Omron CX-Programmer project NewProject (CX-Programmer 9.74)

# PLC GERAL: CJ2M CPU33
I/O table (CPU CJ2M-CPU33): rack 0 slot 0 CJ1W-SCU21; rack 0 slot 1 CJ1W-DRM21; rack 0 slot 2 CJ1W-ID211; rack 0 slot 3 CJ1W-OC211; rack 0 slot 4 CJ1W-MAD42; rack 0 slot 11 CJ2M-EIP21

## Data types
TYPE s_equip_ios : STRUCT  (* Equipamento - Entradas *)
  om : BOOL;  (* Ordem de marcha *)
  oma : BOOL;  (* Ordem de abrir *)
  omf : BOOL;  (* Ordem de fechar *)
  rm : BOOL;  (* Resposta de marcha *)
  fca : BOOL;  (* Fim de curso aberta *)
  fcf : BOOL;  (* Fim de curso fechada *)
  de : BOOL;  (* Defeito electrico *)
  pf_bmb : BOOL;  (* Pulsos de funcionamento da bomba *)
END_STRUCT END_TYPE
TYPE s_equip_bits : STRUCT  (* Equipamento - Bits auxiliares *)
  s_aut : BOOL;  (* Automatico *)
  mdp : BOOL;  (* Disponibilidade *)
  ndp : BOOL;  (* Não disponivel *)
  dgm : BOOL;  (* Defeito geral de maquina *)
  rst : BOOL;  (* Reset *)
  cfa : BOOL;  (* Condição de funcionamento automatico *)
  cfm : BOOL;  (* Condição de funcionamento manual *)
  cfaa : BOOL;  (* Condição de funcionamento automatico abrir *)
  cfaf : BOOL;  (* Condição de funcionamento automatico fechar *)
  cfma : BOOL;  (* Condição de funcionamento manual abrir *)
  cfmf : BOOL;  (* Condição de funcionamento manual fechar *)
  st_hmi : BOOL;  (* Arranque HMI *)
  sp_hmi : BOOL;  (* Paragem HMI *)
  p_hmi : BOOL;  (* Pausa HMI *)
END_STRUCT END_TYPE
TYPE s_equip_defs : STRUCT  (* Equipamentos - Defeitos *)
  fm : BOOL;  (* Falha de marcha *)
  fma : BOOL;  (* Falha de manobra abrir *)
  fmf : BOOL;  (* Falha de manobra fechar *)
  de : BOOL;  (* Defeito electrico *)
  dv : BOOL;  (* Deposito vazio *)
END_STRUCT END_TYPE
TYPE s_equip : STRUCT  (* Equipamento *)
  ios : s_equip_ios;  (* Entradas *)
  bits : s_equip_bits;  (* Bits *)
  defs : s_equip_defs;  (* Defeitos *)
  es : INT;  (* Estado *)
  tm_b : INT;  (* Tempo entre bombagens *)
  rsv1 : INT Dimensions=[5];  (* Reserva *)
END_STRUCT END_TYPE
TYPE s_deposito_p : STRUCT  (* Deposito de produto *)
  prod : INT;  (* Produto *)
  s_aut : BOOL;  (* Automatico *)
  mdp : BOOL;  (* Disponibilidade *)
  ndp : BOOL;  (* Não disponivel *)
  dgm : BOOL;  (* Defeito geral de maquina *)
  rst : BOOL;  (* Reset *)
  on : BOOL;  (* Deposito ligado *)
  oms_red : BOOL;  (* Lampada FLASH vermelho *)
  oms_green : BOOL;  (* Lampada FLASH verde *)
  rsv1 : INT Dimensions=[8];  (* Reserva *)
END_STRUCT END_TYPE
TYPE s_caudal : STRUCT  (* Dados do caudalimetro *)
  tti : BOOL;  (* Impulso de totalização *)
  rst : BOOL;  (* Reset *)
  prod_used : BOOL;  (* Produto em uso *)
  fgp : BOOL;  (* Fuga de produto *)
  ftt : BOOL;  (* Falha de caudal *)
  rem : BOOL;  (* Totalizador local/remoto *)
  rem_ok : BOOL;  (* OK para ir buscar o valor do totalizador remoto *)
  inj_ini : BOOL;  (* Inicio da injecção *)
  x0_8 : BOOL;  (* RESERVA *)
  x0_9 : BOOL;  (* RESERVA *)
  x0_10 : BOOL;  (* RESERVA *)
  x0_11 : BOOL;  (* RESERVA *)
  x0_12 : BOOL;  (* RESERVA *)
  x0_13 : BOOL;  (* RESERVA *)
  x0_14 : BOOL;  (* RESERVA *)
  x0_15 : BOOL;  (* RESERVA *)
  prod : INT;  (* Produto *)
  rsv1 : INT Dimensions=[6];  (* RESERVA *)
  tti_x : REAL;  (* Valor do impulso *)
  tt_rem : REAL;  (* Totalizador remoto *)
  tt_rem_old : REAL;  (* Totalizador remoto antigo *)
  tt_inj : REAL;  (* Totalizador de injecção *)
  tt_p : REAL;  (* Totalizador parcial *)
  tt_g : REAL;  (* Totalizador global *)
END_STRUCT END_TYPE
TYPE s_relogio : STRUCT  (* Dados de acerto e leitura de relógio *)
  pc_ano : INT;  (* Ano *)
  pc_mes : INT;  (* Mes *)
  pc_dia : INT;  (* Dia *)
  pc_dia_s : INT;  (* Dia da semana *)
  pc_hora : INT;  (* Hora *)
  pc_minuto : INT;  (* Minuto *)
  pc_segundo : INT;  (* Segundo *)
  rsv1 : INT Dimensions=[3];  (* RESERVA *)
  ano : INT;  (* Ano *)
  mes : INT;  (* Mes *)
  dia : INT;  (* Dia *)
  dia_s : INT;  (* Dia da semana *)
  hora : INT;  (* Hora *)
  minuto : INT;  (* Minuto *)
  segundo : INT;  (* Segundo *)
  rsv2 : INT Dimensions=[3];  (* RESERVA *)
END_STRUCT END_TYPE

## Global symbols (name address type ; comment)
D10103.00 BOOL  ; 3
fb_dp_bmb_DP03 fb_dp_bmb
fb_dp_bmb_DP04 fb_dp_bmb
fb_dp_bmb_agi_DP05 fb_dp_bmb_agi
fb_dp_pss_agi_vlv_DP01 fb_dp_pss_agi_vlv
fb_dp_pss_agi_vlv_DP02 fb_dp_pss_agi_vlv
fb_eq_agitador_DP01 fb_eq_motor
fb_eq_agitador_DP02 fb_eq_motor
fb_eq_agitador_DP05 fb_eq_motor
fb_eq_bomba_DP03 fb_eq_bomba
fb_eq_bomba_DP04 fb_eq_bomba
fb_eq_bomba_DP05 fb_eq_bomba
fb_eq_press_DP01 fb_eq_press
fb_eq_press_DP02 fb_eq_press
fb_eq_valvula_DP01 fb_eq_valvula
fb_eq_valvula_DP02 fb_eq_valvula
fb_inj_caudal_DP01 fb_inj_caudal
fb_inj_caudal_DP02 fb_inj_caudal
fb_inj_caudal_DP03 fb_inj_caudal
fb_inj_caudal_DP04 fb_inj_caudal
fb_inj_caudal_DP05 fb_inj_caudal
fb_prod_ok fb_prod_ok

## Program Geral (cyclic task 0)
Local symbols
de_agi 0.08 BOOL  ; Termicos Agitadores Parafina/TR02/Teflon
dp01 D0 STRUCT s_deposito_p  ; Deposito de parafina
dp01_agi D20 STRUCT s_equip  ; Agitador de parafina
dp01_pss D10 STRUCT s_equip  ; Presseorização de parafina
dp01_vlv D30 STRUCT s_equip  ; Valvula de parafina
dp02 D100 STRUCT s_deposito_p  ; Deposito de silicone
dp02_agi D120 STRUCT s_equip  ; Agitador de silicone
dp02_pss D110 STRUCT s_equip  ; Presseorização de silicone
dp02_vlv D130 STRUCT s_equip  ; Valvula de silicone
dp03 D200 STRUCT s_deposito_p  ; Deposito de caf
dp03_bmb D210 STRUCT s_equip  ; Bomba de caf
dp04 D300 STRUCT s_deposito_p  ; Deposito de bopsil
dp04_bmb D310 STRUCT s_equip  ; Bomba de bopsil
dp05 D400 STRUCT s_deposito_p  ; Deposito de teflon
dp05_agi D420 STRUCT s_equip  ; Agitador de teflon
dp05_bmb D410 STRUCT s_equip  ; Bomba de teflon
m_prod_in W100 INT[10]  ; Pedidos de produto das maquinas
m_prod_out D10010 INT[10]  ; Autorização de produto para as maquinas
om_a_p2x 1.02 BOOL  ; Agitador P2X
om_a_parafina 1.00 BOOL  ; Agitador PARAFINA
om_a_tr02 1.01 BOOL  ; Agitador TR02
om_b_bopsil 1.14 BOOL  ; Bomba BOPSIL
om_b_caf 1.07 BOOL  ; Bomba CAF
om_b_p2x 1.13 BOOL  ; Bomba P2X
om_p_parafina 1.05 BOOL  ; Pressuriza Dep.PARAFINA
om_p_tr02 1.06 BOOL  ; Pressuriza Dep.TR02
oma_v_parafina 1.11 BOOL  ; Valvula Saida Dep PARAFINA
oma_v_tr02 1.12 BOOL  ; Valvula Saida Dep TR02
oms_alarm 1.08 BOOL  ; FLASH alarme
pe_geral 0.00 BOOL  ; Emergencia Geral
pf_bopsil 0.10 BOOL  ; Sensor bomba BOPSIL
pf_caf 0.09 BOOL  ; Sensor bomba CAF
pf_p2x 0.11 BOOL  ; Sensor bomba P2X
prod_used D10009.00 BOOL[10]  ; Produto em uso
psl_geral 0.06 BOOL  ; Presssostato
rm_geral 0.07 BOOL  ; Confirmação Despoeiramento
tt_dp01 D600 STRUCT s_caudal  ; Caudalímetro de bopsil
tt_dp02 D620 STRUCT s_caudal  ; Caudalímetro de caf
tt_dp03 D640 STRUCT s_caudal  ; Caudalímetro de teflon
tt_dp04 D660 STRUCT s_caudal  ; Caudalímetro de paradina
tt_dp05 D680 STRUCT s_caudal  ; Caudalímetro de tr02
tti_bopsil 0.04 BOOL  ; Caudalimetro BOPSIL
tti_caf 0.03 BOOL  ; Caudalimetro CAF
tti_p2x 0.05 BOOL  ; Caudalimetro P2X
tti_parafina 0.01 BOOL  ; Caudalimetro PARAFINA
tti_tr02 0.02 BOOL  ; Caudalimetro TR02

### Section PARAFINA

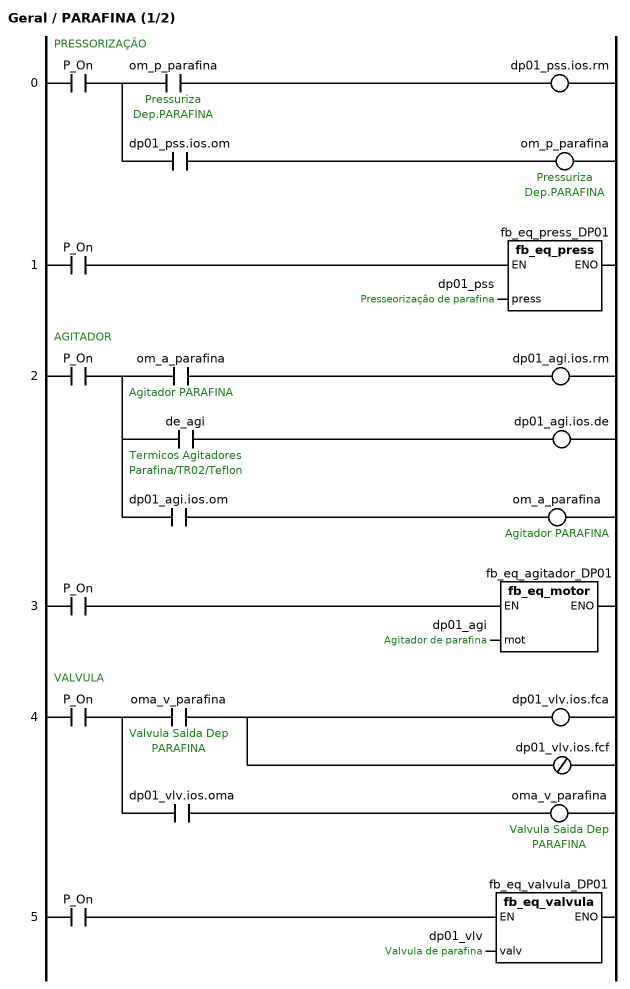
; rung 0: PRESSORIZAÇÃO
LD P_On
OUT TR0
AND om_p_parafina  ; Pressuriza Dep.PARAFINA
OUT dp01_pss.ios.rm
LD TR0
AND dp01_pss.ios.om
OUT om_p_parafina  ; Pressuriza Dep.PARAFINA
; rung 1
LD P_On
CALL fb_eq_press_DP01 : fb_eq_press (press := dp01_pss)  ; Presseorização de parafina
; rung 2: AGITADOR
LD P_On
OUT TR0
AND om_a_parafina  ; Agitador PARAFINA
OUT dp01_agi.ios.rm
LD TR0
AND de_agi  ; Termicos Agitadores Parafina/TR02/Teflon
OUT dp01_agi.ios.de
LD TR0
AND dp01_agi.ios.om
OUT om_a_parafina  ; Agitador PARAFINA
; rung 3
LD P_On
CALL fb_eq_agitador_DP01 : fb_eq_motor (mot := dp01_agi)  ; Agitador de parafina
; rung 4: VALVULA
LD P_On
OUT TR0
AND oma_v_parafina  ; Valvula Saida Dep PARAFINA
OUT dp01_vlv.ios.fca
OUTNOT dp01_vlv.ios.fcf
LD TR0
AND dp01_vlv.ios.oma
OUT oma_v_parafina  ; Valvula Saida Dep PARAFINA
; rung 5
LD P_On
CALL fb_eq_valvula_DP01 : fb_eq_valvula (valv := dp01_vlv)  ; Valvula de parafina

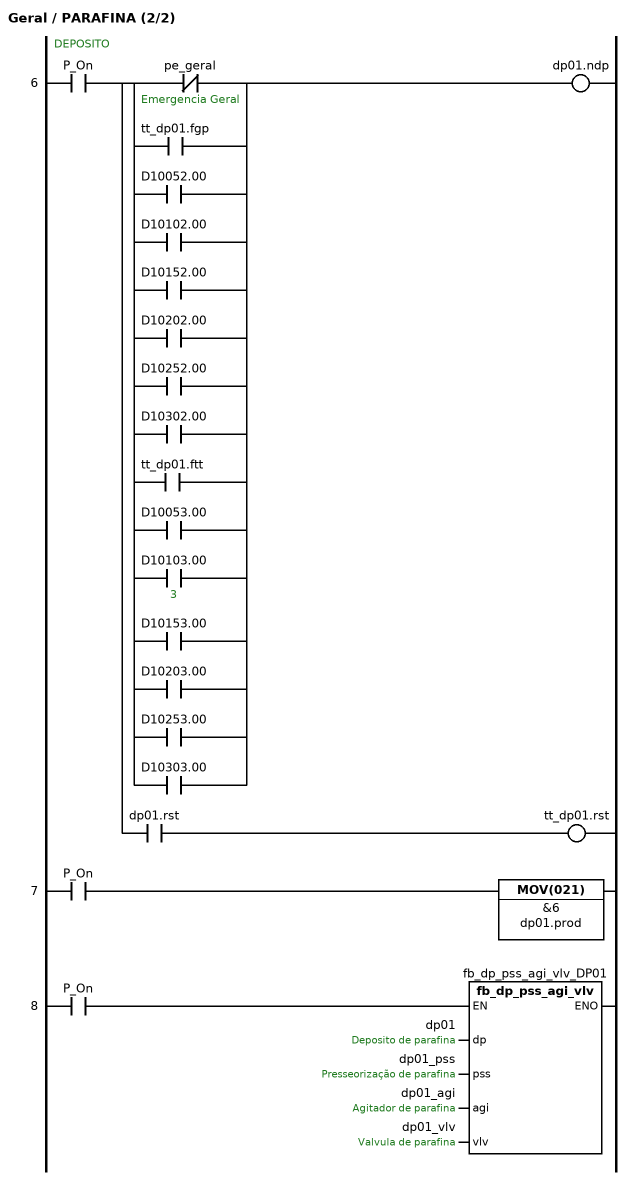
; rung 6: DEPOSITO
LD P_On
OUT TR0
LDNOT pe_geral  ; Emergencia Geral
OR tt_dp01.fgp
OR D10052.00
OR D10102.00
OR D10152.00
OR D10202.00
OR D10252.00
OR D10302.00
OR tt_dp01.ftt
OR D10053.00
OR D10103.00  ; 3
OR D10153.00
OR D10203.00
OR D10253.00
OR D10303.00
ANDLD
OUT dp01.ndp
LD TR0
AND dp01.rst
OUT tt_dp01.rst
; rung 7
LD P_On
MOV(021) &6 dp01.prod
; rung 8
LD P_On
CALL fb_dp_pss_agi_vlv_DP01 : fb_dp_pss_agi_vlv (dp := dp01, pss := dp01_pss, agi := dp01_agi, vlv := dp01_vlv)  ; Deposito de parafina, Presseorização de parafina, Agitador de parafina, Valvula de parafina

### Section SILICONE_TR02

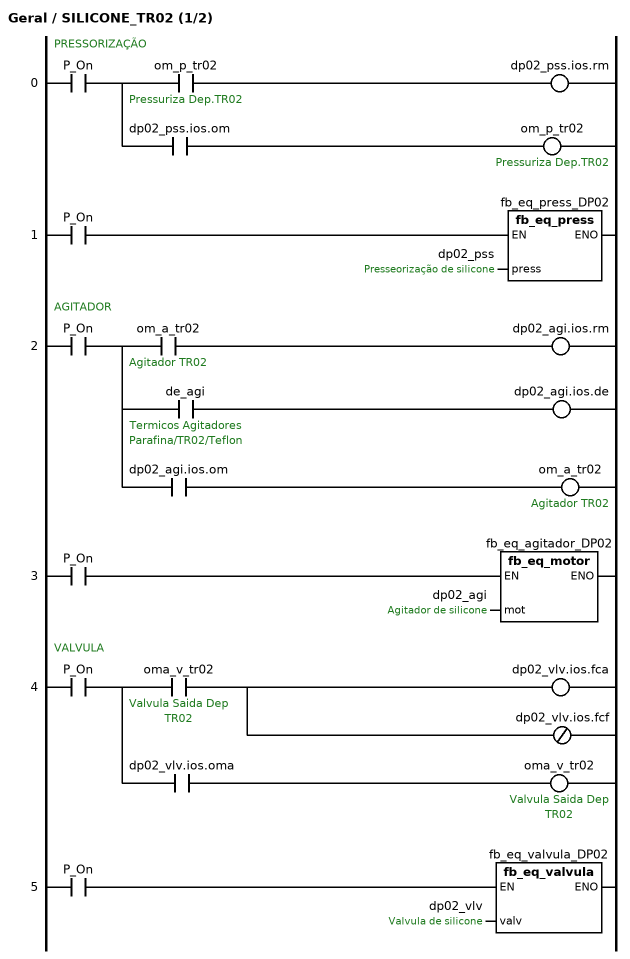
; rung 0: PRESSORIZAÇÃO
LD P_On
OUT TR0
AND om_p_tr02  ; Pressuriza Dep.TR02
OUT dp02_pss.ios.rm
LD TR0
AND dp02_pss.ios.om
OUT om_p_tr02  ; Pressuriza Dep.TR02
; rung 1
LD P_On
CALL fb_eq_press_DP02 : fb_eq_press (press := dp02_pss)  ; Presseorização de silicone
; rung 2: AGITADOR
LD P_On
OUT TR0
AND om_a_tr02  ; Agitador TR02
OUT dp02_agi.ios.rm
LD TR0
AND de_agi  ; Termicos Agitadores Parafina/TR02/Teflon
OUT dp02_agi.ios.de
LD TR0
AND dp02_agi.ios.om
OUT om_a_tr02  ; Agitador TR02
; rung 3
LD P_On
CALL fb_eq_agitador_DP02 : fb_eq_motor (mot := dp02_agi)  ; Agitador de silicone
; rung 4: VALVULA
LD P_On
OUT TR0
AND oma_v_tr02  ; Valvula Saida Dep TR02
OUT dp02_vlv.ios.fca
OUTNOT dp02_vlv.ios.fcf
LD TR0
AND dp02_vlv.ios.oma
OUT oma_v_tr02  ; Valvula Saida Dep TR02
; rung 5
LD P_On
CALL fb_eq_valvula_DP02 : fb_eq_valvula (valv := dp02_vlv)  ; Valvula de silicone

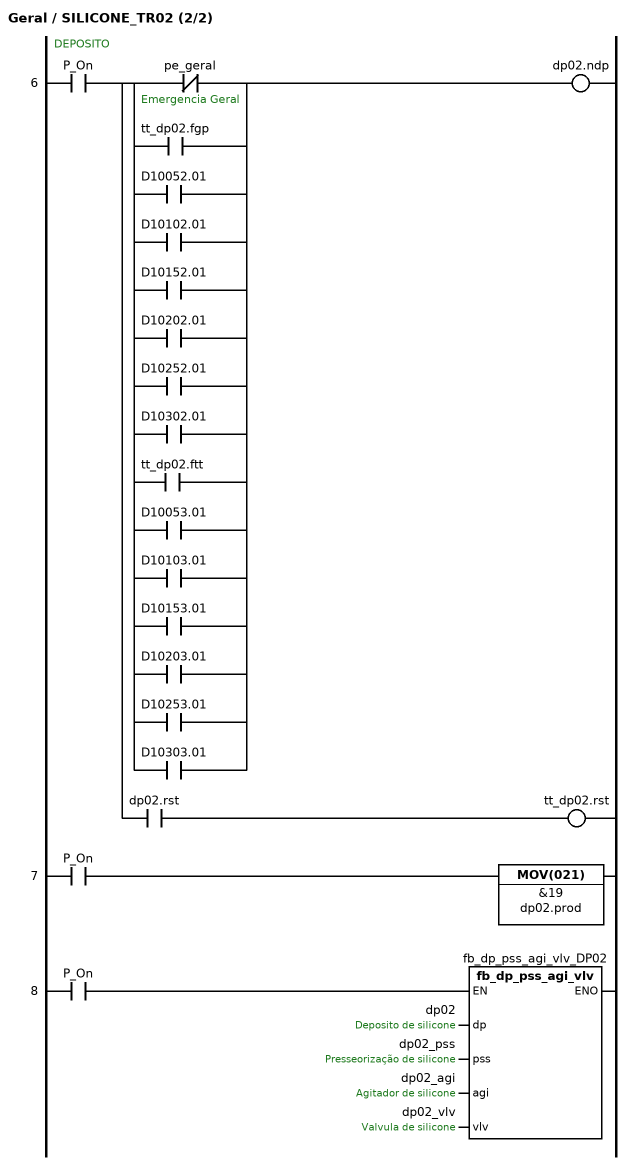
; rung 6: DEPOSITO
LD P_On
OUT TR0
LDNOT pe_geral  ; Emergencia Geral
OR tt_dp02.fgp
OR D10052.01
OR D10102.01
OR D10152.01
OR D10202.01
OR D10252.01
OR D10302.01
OR tt_dp02.ftt
OR D10053.01
OR D10103.01
OR D10153.01
OR D10203.01
OR D10253.01
OR D10303.01
ANDLD
OUT dp02.ndp
LD TR0
AND dp02.rst
OUT tt_dp02.rst
; rung 7
LD P_On
MOV(021) &19 dp02.prod
; rung 8
LD P_On
CALL fb_dp_pss_agi_vlv_DP02 : fb_dp_pss_agi_vlv (dp := dp02, pss := dp02_pss, agi := dp02_agi, vlv := dp02_vlv)  ; Deposito de silicone, Presseorização de silicone, Agitador de silicone, Valvula de silicone

### Section CAF

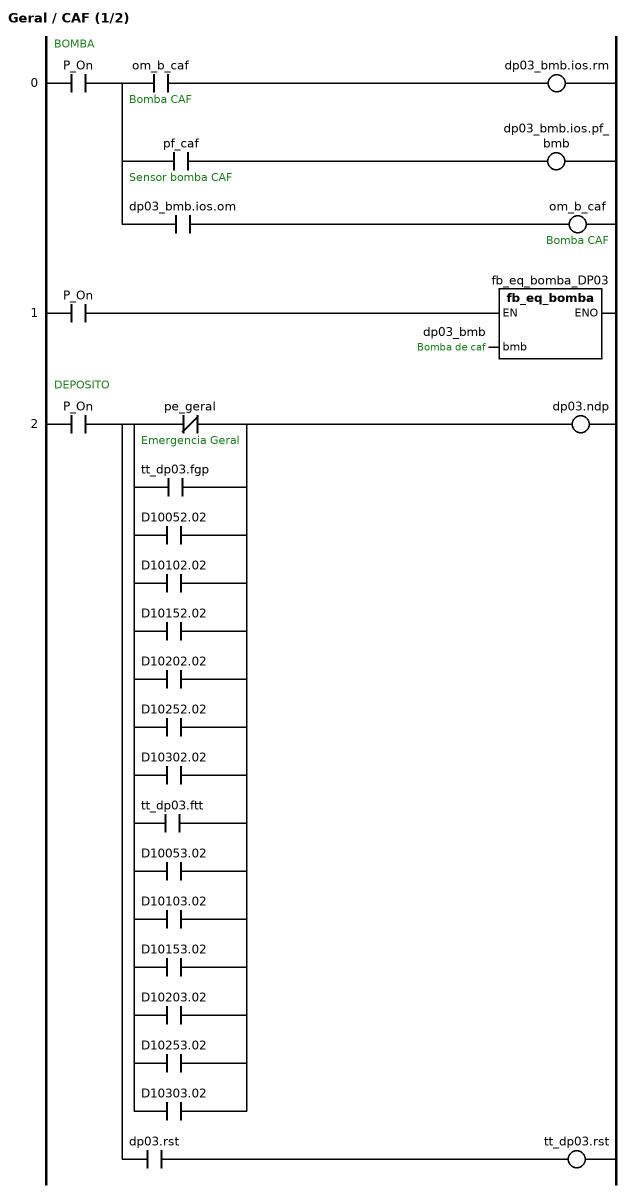
; rung 0: BOMBA
LD P_On
OUT TR0
AND om_b_caf  ; Bomba CAF
OUT dp03_bmb.ios.rm
LD TR0
AND pf_caf  ; Sensor bomba CAF
OUT dp03_bmb.ios.pf_bmb
LD TR0
AND dp03_bmb.ios.om
OUT om_b_caf  ; Bomba CAF
; rung 1
LD P_On
CALL fb_eq_bomba_DP03 : fb_eq_bomba (bmb := dp03_bmb)  ; Bomba de caf
; rung 2: DEPOSITO
LD P_On
OUT TR0
LDNOT pe_geral  ; Emergencia Geral
OR tt_dp03.fgp
OR D10052.02
OR D10102.02
OR D10152.02
OR D10202.02
OR D10252.02
OR D10302.02
OR tt_dp03.ftt
OR D10053.02
OR D10103.02
OR D10153.02
OR D10203.02
OR D10253.02
OR D10303.02
ANDLD
OUT dp03.ndp
LD TR0
AND dp03.rst
OUT tt_dp03.rst

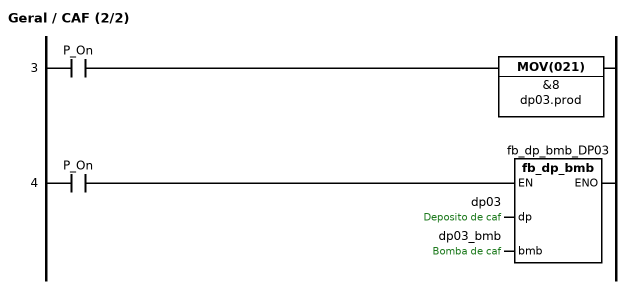
; rung 3
LD P_On
MOV(021) &8 dp03.prod
; rung 4
LD P_On
CALL fb_dp_bmb_DP03 : fb_dp_bmb (dp := dp03, bmb := dp03_bmb)  ; Deposito de caf, Bomba de caf

### Section BOPSIL

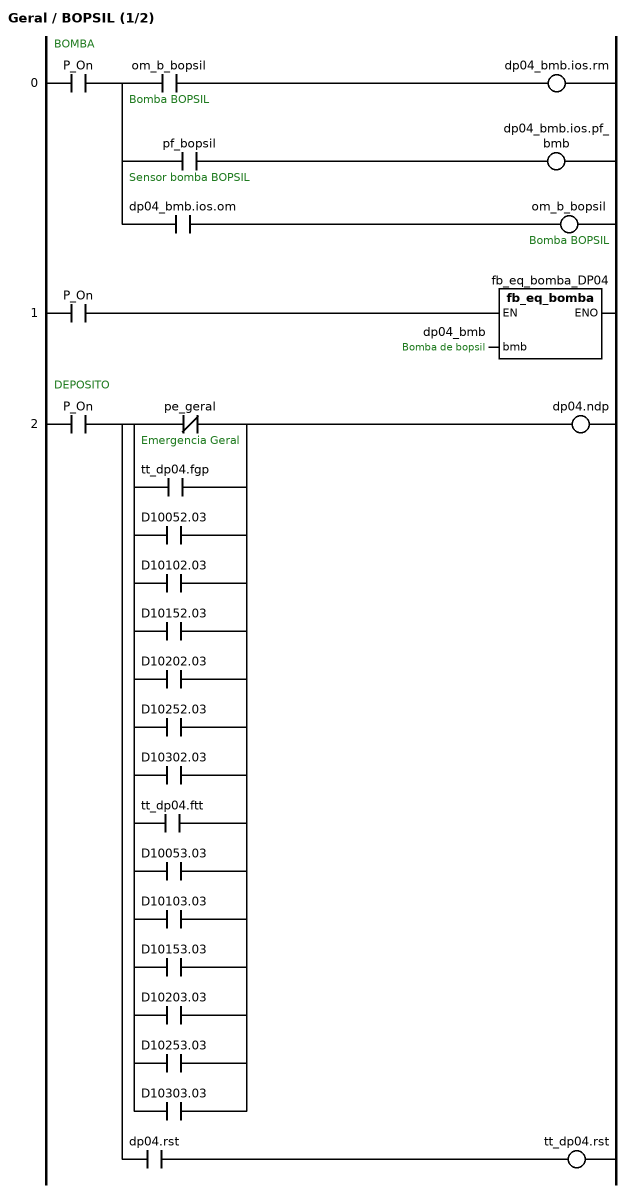
; rung 0: BOMBA
LD P_On
OUT TR0
AND om_b_bopsil  ; Bomba BOPSIL
OUT dp04_bmb.ios.rm
LD TR0
AND pf_bopsil  ; Sensor bomba BOPSIL
OUT dp04_bmb.ios.pf_bmb
LD TR0
AND dp04_bmb.ios.om
OUT om_b_bopsil  ; Bomba BOPSIL
; rung 1
LD P_On
CALL fb_eq_bomba_DP04 : fb_eq_bomba (bmb := dp04_bmb)  ; Bomba de bopsil
; rung 2: DEPOSITO
LD P_On
OUT TR0
LDNOT pe_geral  ; Emergencia Geral
OR tt_dp04.fgp
OR D10052.03
OR D10102.03
OR D10152.03
OR D10202.03
OR D10252.03
OR D10302.03
OR tt_dp04.ftt
OR D10053.03
OR D10103.03
OR D10153.03
OR D10203.03
OR D10253.03
OR D10303.03
ANDLD
OUT dp04.ndp
LD TR0
AND dp04.rst
OUT tt_dp04.rst

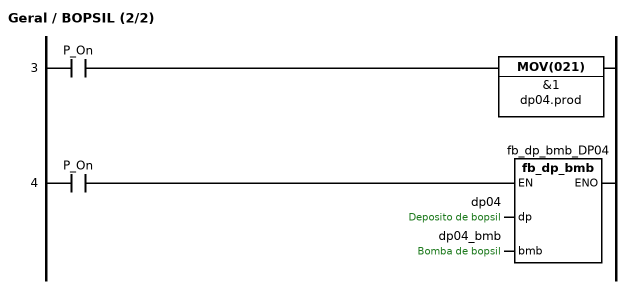
; rung 3
LD P_On
MOV(021) &1 dp04.prod
; rung 4
LD P_On
CALL fb_dp_bmb_DP04 : fb_dp_bmb (dp := dp04, bmb := dp04_bmb)  ; Deposito de bopsil, Bomba de bopsil

### Section LUBCORK_P2X

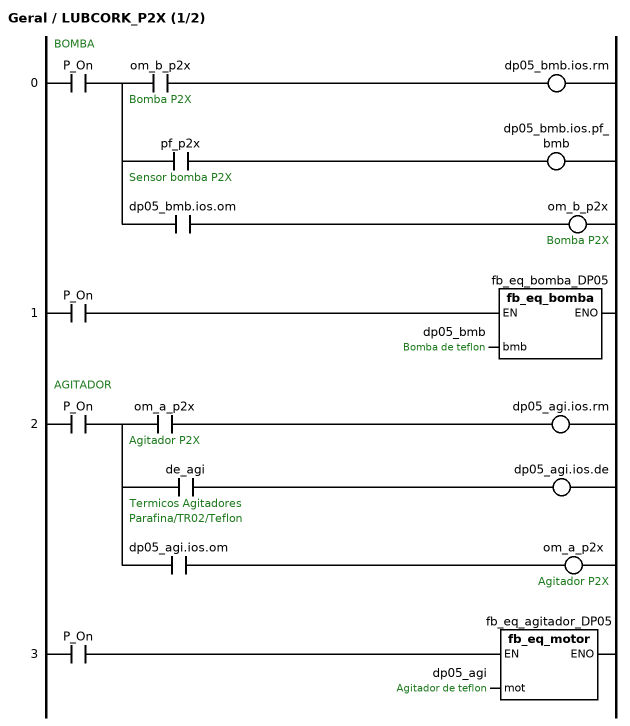
; rung 0: BOMBA
LD P_On
OUT TR0
AND om_b_p2x  ; Bomba P2X
OUT dp05_bmb.ios.rm
LD TR0
AND pf_p2x  ; Sensor bomba P2X
OUT dp05_bmb.ios.pf_bmb
LD TR0
AND dp05_bmb.ios.om
OUT om_b_p2x  ; Bomba P2X
; rung 1
LD P_On
CALL fb_eq_bomba_DP05 : fb_eq_bomba (bmb := dp05_bmb)  ; Bomba de teflon
; rung 2: AGITADOR
LD P_On
OUT TR0
AND om_a_p2x  ; Agitador P2X
OUT dp05_agi.ios.rm
LD TR0
AND de_agi  ; Termicos Agitadores Parafina/TR02/Teflon
OUT dp05_agi.ios.de
LD TR0
AND dp05_agi.ios.om
OUT om_a_p2x  ; Agitador P2X
; rung 3
LD P_On
CALL fb_eq_agitador_DP05 : fb_eq_motor (mot := dp05_agi)  ; Agitador de teflon

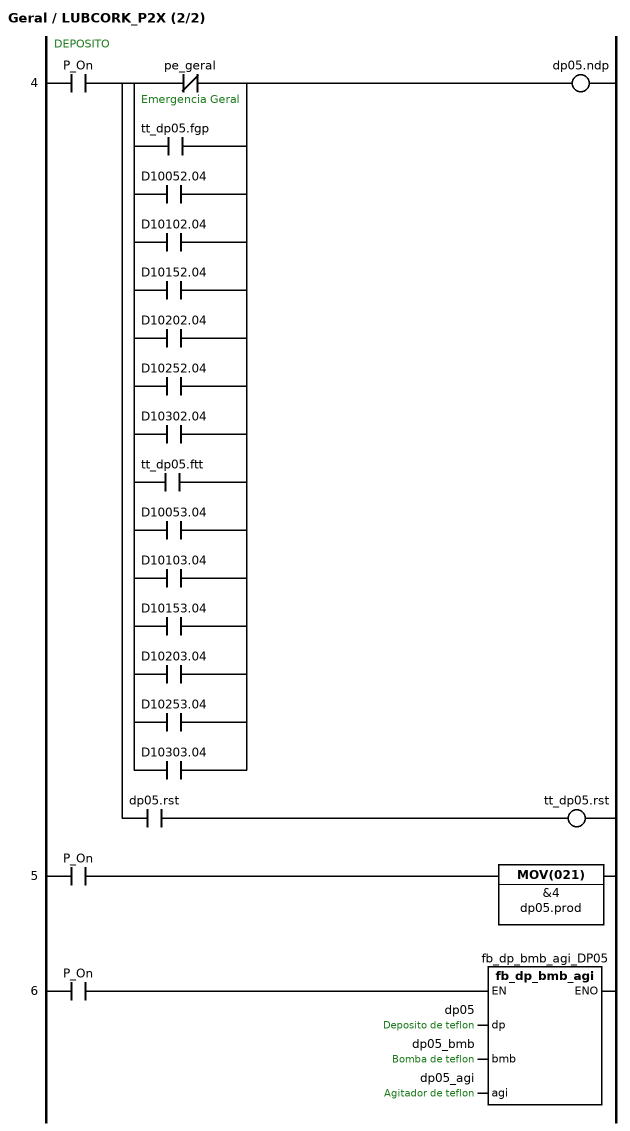
; rung 4: DEPOSITO
LD P_On
OUT TR0
LDNOT pe_geral  ; Emergencia Geral
OR tt_dp05.fgp
OR D10052.04
OR D10102.04
OR D10152.04
OR D10202.04
OR D10252.04
OR D10302.04
OR tt_dp05.ftt
OR D10053.04
OR D10103.04
OR D10153.04
OR D10203.04
OR D10253.04
OR D10303.04
ANDLD
OUT dp05.ndp
LD TR0
AND dp05.rst
OUT tt_dp05.rst
; rung 5
LD P_On
MOV(021) &4 dp05.prod
; rung 6
LD P_On
CALL fb_dp_bmb_agi_DP05 : fb_dp_bmb_agi (dp := dp05, bmb := dp05_bmb, agi := dp05_agi)  ; Deposito de teflon, Bomba de teflon, Agitador de teflon

### Section CAUDAL

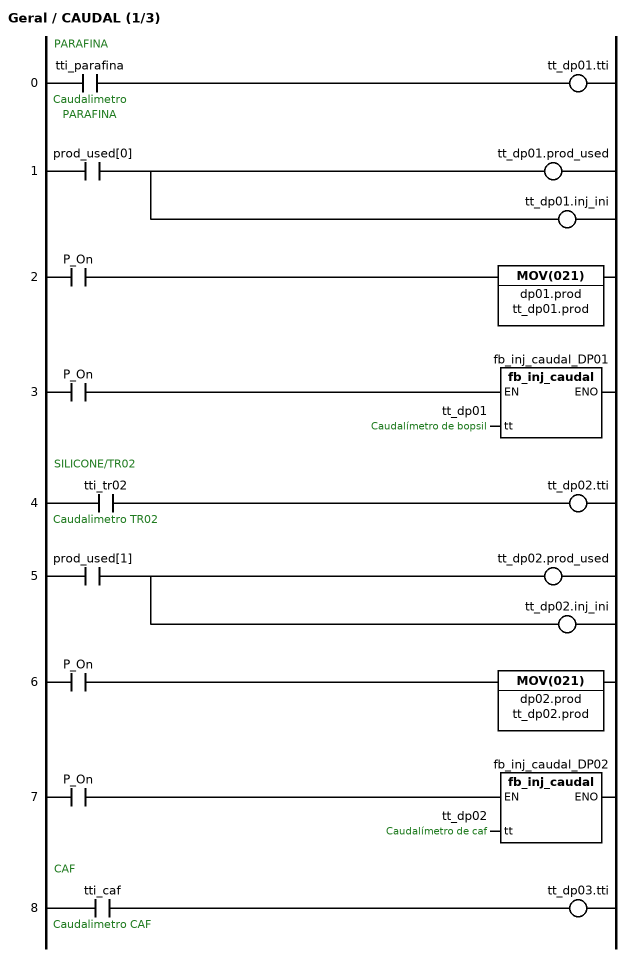
; rung 0: PARAFINA
LD tti_parafina  ; Caudalimetro PARAFINA
OUT tt_dp01.tti
; rung 1
LD prod_used[0]
OUT tt_dp01.prod_used
OUT tt_dp01.inj_ini
; rung 2
LD P_On
MOV(021) dp01.prod tt_dp01.prod
; rung 3
LD P_On
CALL fb_inj_caudal_DP01 : fb_inj_caudal (tt := tt_dp01)  ; Caudalímetro de bopsil
; rung 4: SILICONE/TR02
LD tti_tr02  ; Caudalimetro TR02
OUT tt_dp02.tti
; rung 5
LD prod_used[1]
OUT tt_dp02.prod_used
OUT tt_dp02.inj_ini
; rung 6
LD P_On
MOV(021) dp02.prod tt_dp02.prod
; rung 7
LD P_On
CALL fb_inj_caudal_DP02 : fb_inj_caudal (tt := tt_dp02)  ; Caudalímetro de caf
; rung 8: CAF
LD tti_caf  ; Caudalimetro CAF
OUT tt_dp03.tti

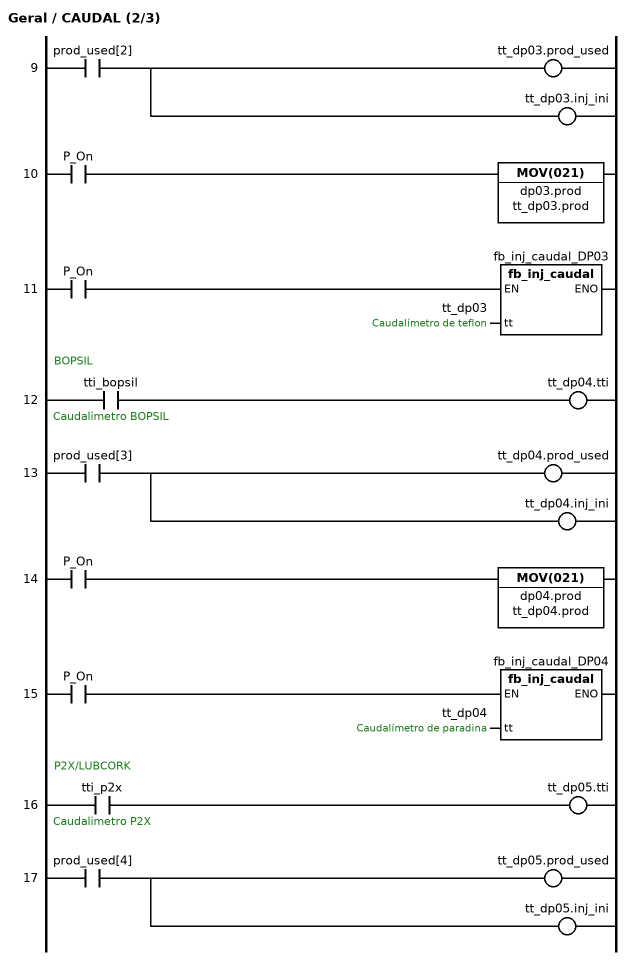
; rung 9
LD prod_used[2]
OUT tt_dp03.prod_used
OUT tt_dp03.inj_ini
; rung 10
LD P_On
MOV(021) dp03.prod tt_dp03.prod
; rung 11
LD P_On
CALL fb_inj_caudal_DP03 : fb_inj_caudal (tt := tt_dp03)  ; Caudalímetro de teflon
; rung 12: BOPSIL
LD tti_bopsil  ; Caudalimetro BOPSIL
OUT tt_dp04.tti
; rung 13
LD prod_used[3]
OUT tt_dp04.prod_used
OUT tt_dp04.inj_ini
; rung 14
LD P_On
MOV(021) dp04.prod tt_dp04.prod
; rung 15
LD P_On
CALL fb_inj_caudal_DP04 : fb_inj_caudal (tt := tt_dp04)  ; Caudalímetro de paradina
; rung 16: P2X/LUBCORK
LD tti_p2x  ; Caudalimetro P2X
OUT tt_dp05.tti
; rung 17
LD prod_used[4]
OUT tt_dp05.prod_used
OUT tt_dp05.inj_ini

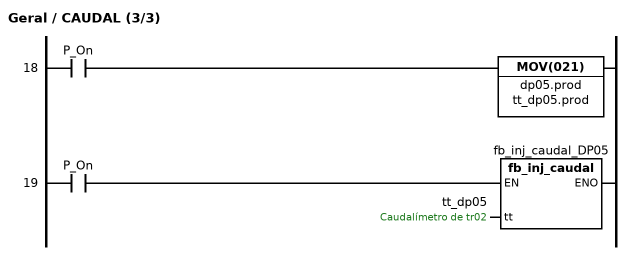
; rung 18
LD P_On
MOV(021) dp05.prod tt_dp05.prod
; rung 19
LD P_On
CALL fb_inj_caudal_DP05 : fb_inj_caudal (tt := tt_dp05)  ; Caudalímetro de tr02

### Section FCOMUNICACAO

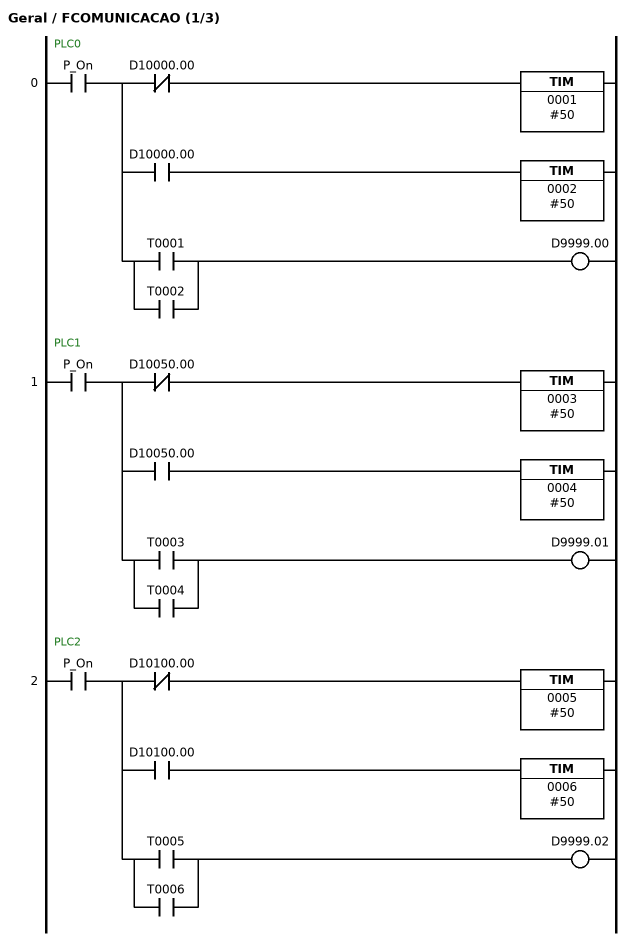
; rung 0: PLC0
LD P_On
OUT TR0
ANDNOT D10000.00
TIM 0001 #50
LD TR0
AND D10000.00
TIM 0002 #50
LD TR0
LD T0001
OR T0002
ANDLD
OUT D9999.00
; rung 1: PLC1
LD P_On
OUT TR0
ANDNOT D10050.00
TIM 0003 #50
LD TR0
AND D10050.00
TIM 0004 #50
LD TR0
LD T0003
OR T0004
ANDLD
OUT D9999.01
; rung 2: PLC2
LD P_On
OUT TR0
ANDNOT D10100.00
TIM 0005 #50
LD TR0
AND D10100.00
TIM 0006 #50
LD TR0
LD T0005
OR T0006
ANDLD
OUT D9999.02

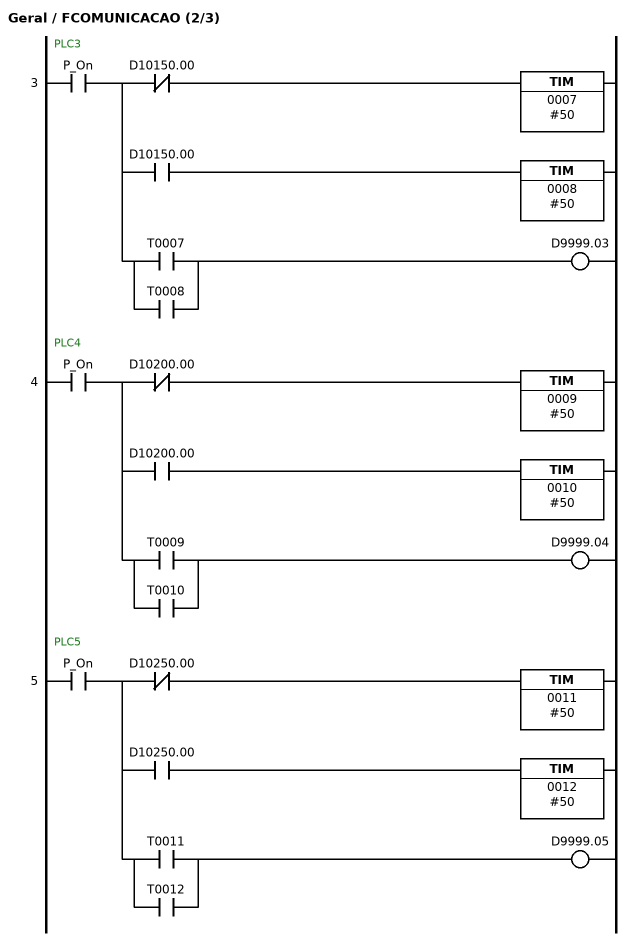
; rung 3: PLC3
LD P_On
OUT TR0
ANDNOT D10150.00
TIM 0007 #50
LD TR0
AND D10150.00
TIM 0008 #50
LD TR0
LD T0007
OR T0008
ANDLD
OUT D9999.03
; rung 4: PLC4
LD P_On
OUT TR0
ANDNOT D10200.00
TIM 0009 #50
LD TR0
AND D10200.00
TIM 0010 #50
LD TR0
LD T0009
OR T0010
ANDLD
OUT D9999.04
; rung 5: PLC5
LD P_On
OUT TR0
ANDNOT D10250.00
TIM 0011 #50
LD TR0
AND D10250.00
TIM 0012 #50
LD TR0
LD T0011
OR T0012
ANDLD
OUT D9999.05

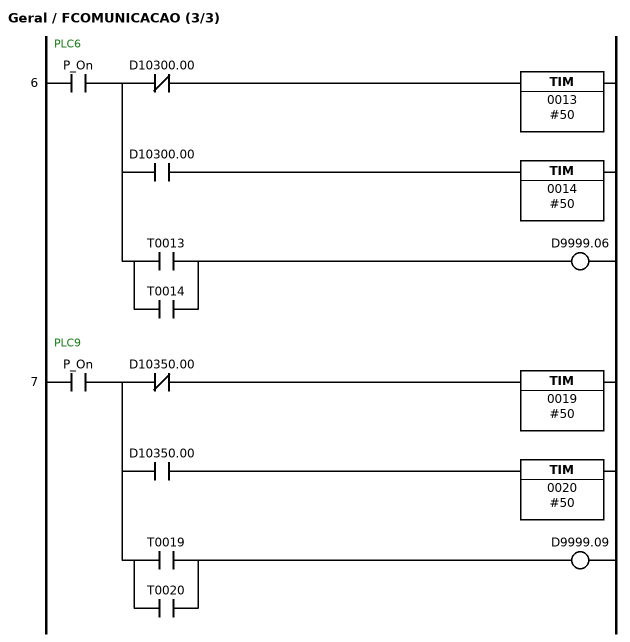
; rung 6: PLC6
LD P_On
OUT TR0
ANDNOT D10300.00
TIM 0013 #50
LD TR0
AND D10300.00
TIM 0014 #50
LD TR0
LD T0013
OR T0014
ANDLD
OUT D9999.06
; rung 7: PLC9
LD P_On
OUT TR0
ANDNOT D10350.00
TIM 0019 #50
LD TR0
AND D10350.00
TIM 0020 #50
LD TR0
LD T0019
OR T0020
ANDLD
OUT D9999.09

### Section COMUNICACAO

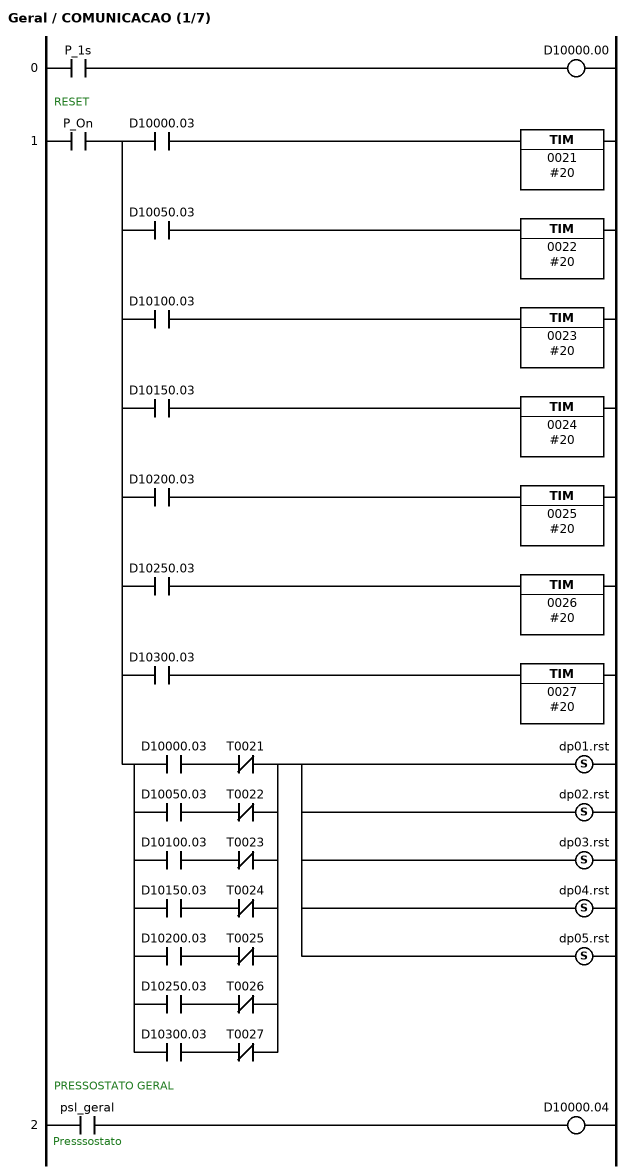
; rung 0
LD P_1s
OUT D10000.00
; rung 1: RESET
LD P_On
OUT TR0
AND D10000.03
TIM 0021 #20
LD TR0
AND D10050.03
TIM 0022 #20
LD TR0
AND D10100.03
TIM 0023 #20
LD TR0
AND D10150.03
TIM 0024 #20
LD TR0
AND D10200.03
TIM 0025 #20
LD TR0
AND D10250.03
TIM 0026 #20
LD TR0
AND D10300.03
TIM 0027 #20
LD TR0
LD D10000.03
ANDNOT T0021
LD D10050.03
ANDNOT T0022
ORLD
LD D10100.03
ANDNOT T0023
ORLD
LD D10150.03
ANDNOT T0024
ORLD
LD D10200.03
ANDNOT T0025
ORLD
LD D10250.03
ANDNOT T0026
ORLD
LD D10300.03
ANDNOT T0027
ORLD
ANDLD
SET dp01.rst
SET dp02.rst
SET dp03.rst
SET dp04.rst
SET dp05.rst
; rung 2: PRESSOSTATO GERAL
LD psl_geral  ; Presssostato
OUT D10000.04

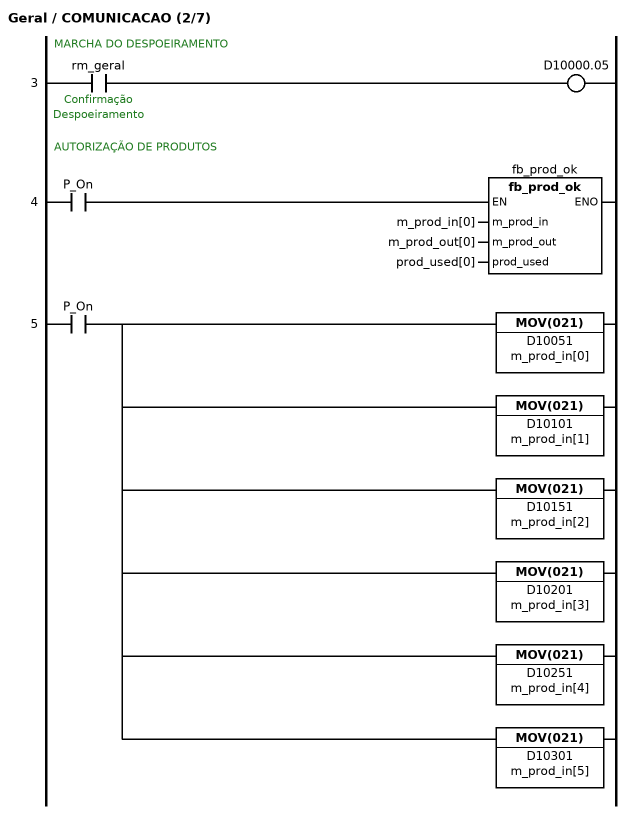
; rung 3: MARCHA DO DESPOEIRAMENTO
LD rm_geral  ; Confirmação Despoeiramento
OUT D10000.05
; rung 4: AUTORIZAÇÃO DE PRODUTOS
LD P_On
CALL fb_prod_ok : fb_prod_ok (m_prod_in := m_prod_in[0], m_prod_out := m_prod_out[0], prod_used := prod_used[0])
; rung 5
LD P_On
MOV(021) D10051 m_prod_in[0]
MOV(021) D10101 m_prod_in[1]
MOV(021) D10151 m_prod_in[2]
MOV(021) D10201 m_prod_in[3]
MOV(021) D10251 m_prod_in[4]
MOV(021) D10301 m_prod_in[5]

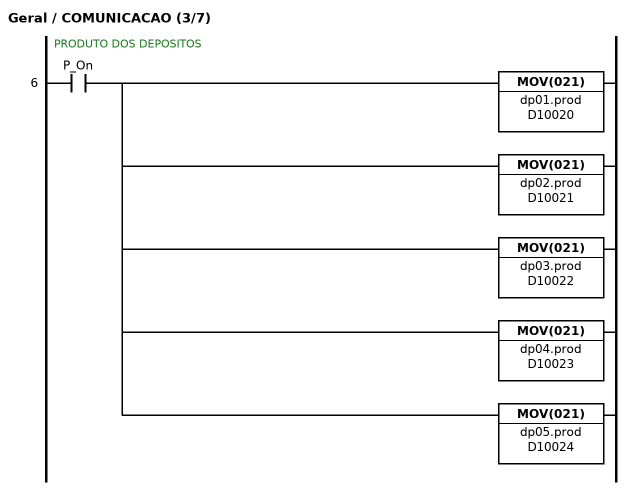
; rung 6: PRODUTO DOS DEPOSITOS
LD P_On
MOV(021) dp01.prod D10020
MOV(021) dp02.prod D10021
MOV(021) dp03.prod D10022
MOV(021) dp04.prod D10023
MOV(021) dp05.prod D10024

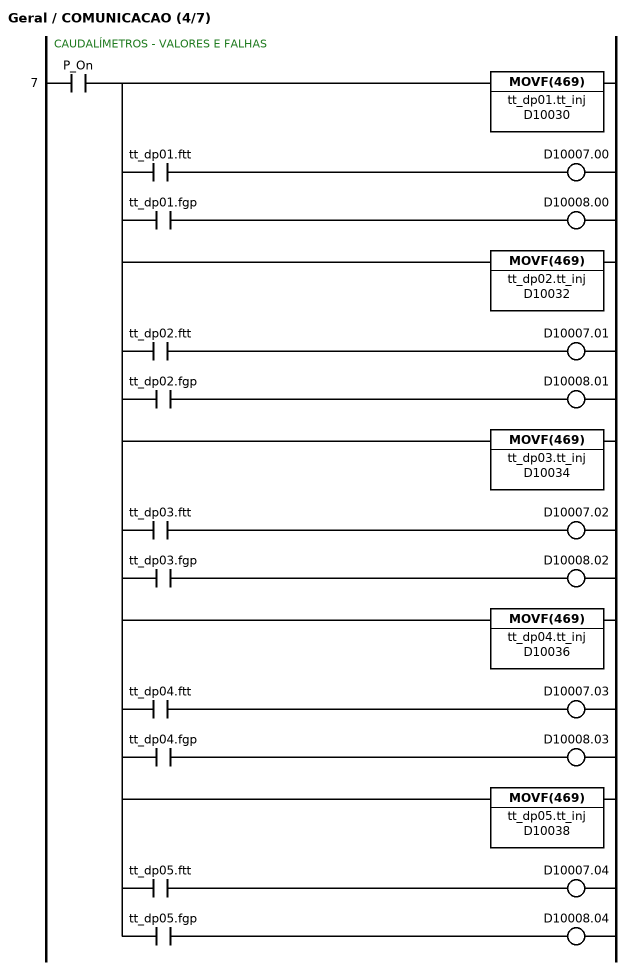
; rung 7: CAUDALÍMETROS - VALORES E FALHAS
LD P_On
OUT TR0
MOVF(469) tt_dp01.tt_inj D10030
AND tt_dp01.ftt
OUT D10007.00
LD TR0
AND tt_dp01.fgp
OUT D10008.00
LD TR0
MOVF(469) tt_dp02.tt_inj D10032
AND tt_dp02.ftt
OUT D10007.01
LD TR0
AND tt_dp02.fgp
OUT D10008.01
LD TR0
MOVF(469) tt_dp03.tt_inj D10034
AND tt_dp03.ftt
OUT D10007.02
LD TR0
AND tt_dp03.fgp
OUT D10008.02
LD TR0
MOVF(469) tt_dp04.tt_inj D10036
AND tt_dp04.ftt
OUT D10007.03
LD TR0
AND tt_dp04.fgp
OUT D10008.03
LD TR0
MOVF(469) tt_dp05.tt_inj D10038
AND tt_dp05.ftt
OUT D10007.04
LD TR0
AND tt_dp05.fgp
OUT D10008.04

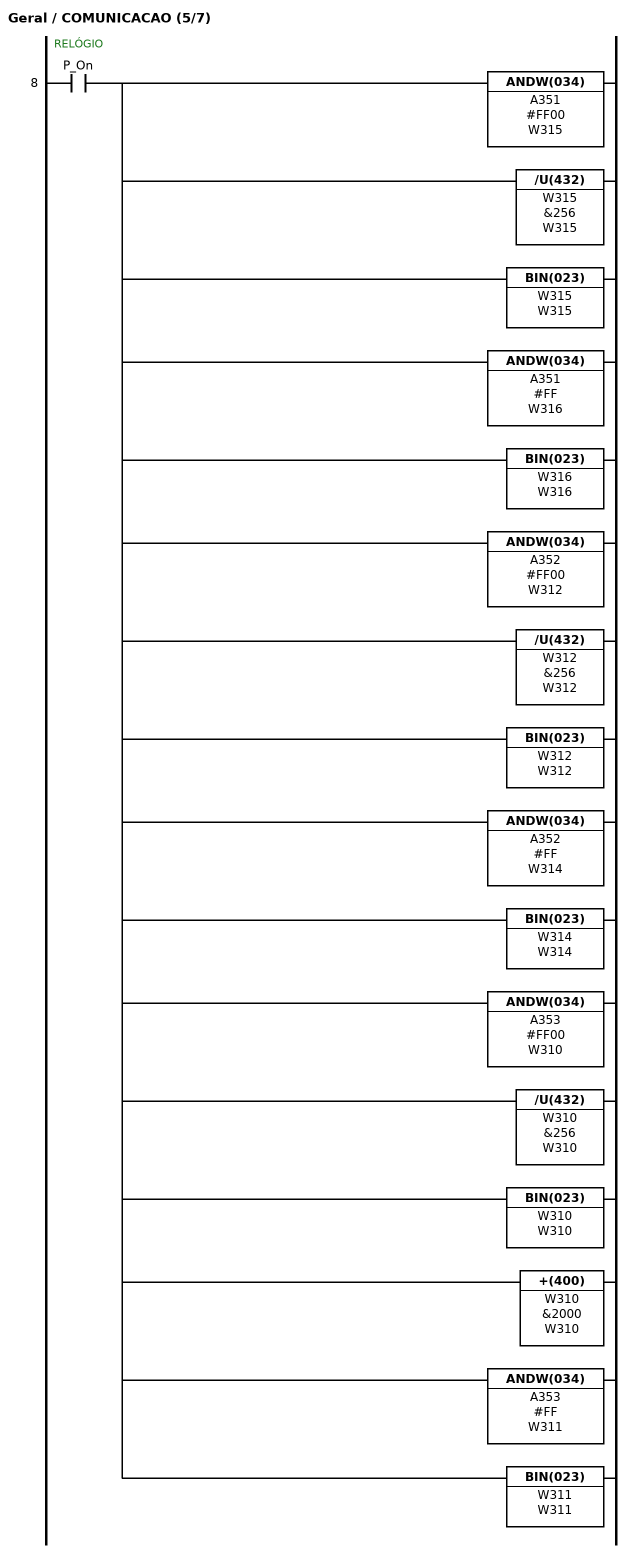
; rung 8: RELÓGIO
LD P_On
ANDW(034) A351 #FF00 W315
/U(432) W315 &256 W315
BIN(023) W315 W315
ANDW(034) A351 #FF W316
BIN(023) W316 W316
ANDW(034) A352 #FF00 W312
/U(432) W312 &256 W312
BIN(023) W312 W312
ANDW(034) A352 #FF W314
BIN(023) W314 W314
ANDW(034) A353 #FF00 W310
/U(432) W310 &256 W310
BIN(023) W310 W310
+(400) W310 &2000 W310
ANDW(034) A353 #FF W311
BIN(023) W311 W311

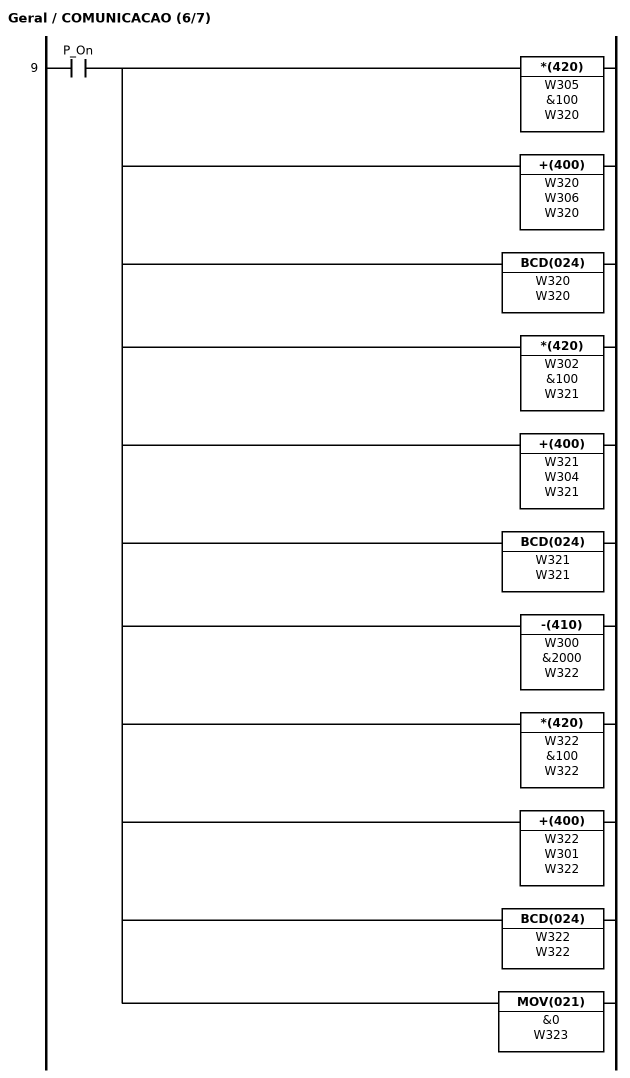
; rung 9
LD P_On
*(420) W305 &100 W320
+(400) W320 W306 W320
BCD(024) W320 W320
*(420) W302 &100 W321
+(400) W321 W304 W321
BCD(024) W321 W321
-(410) W300 &2000 W322
*(420) W322 &100 W322
+(400) W322 W301 W322
BCD(024) W322 W322
MOV(021) &0 W323

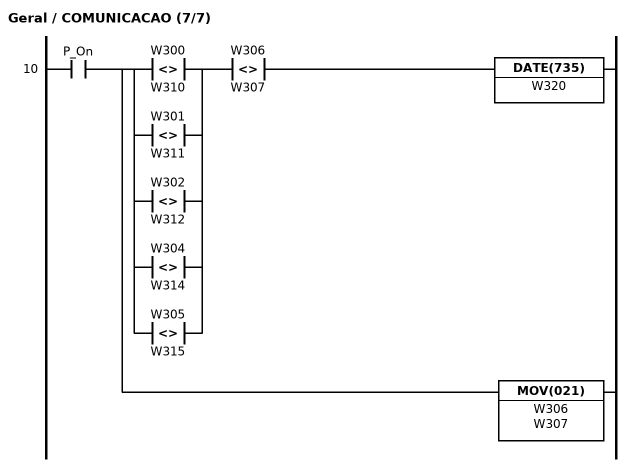
; rung 10
LD P_On
OUT TR0
LD<>(305) W300 W310
OR<>(305) W301 W311
OR<>(305) W302 W312
OR<>(305) W304 W314
OR<>(305) W305 W315
ANDLD
AND<>(305) W306 W307
DATE(735) W320
LD TR0
MOV(021) W306 W307

### Section END
; rung 0
END(001)

## Function block fb_dp_bmb
; FUNÇÃO DEPOSITO DE PRODUTO COM BOMBA - Executa o funcionamento de um deposito de produto constituido apenas por uma bomba.
VAR_IN_OUT
  dp : s_deposito_p;  (* Dados do deposito *)
  bmb : s_equip;  (* Dados da bomba *)
END_VAR

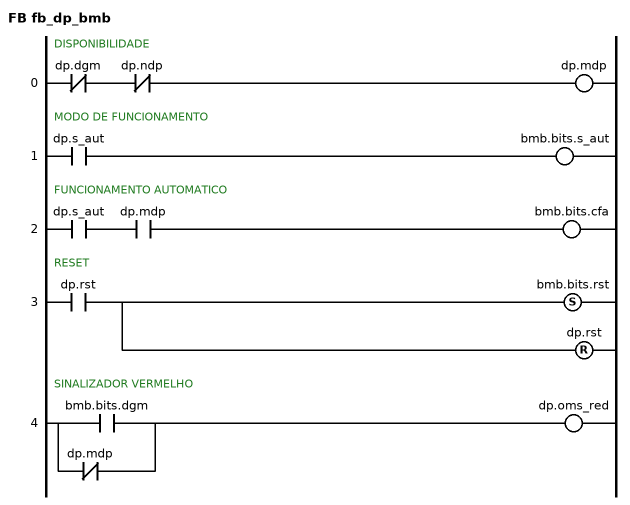
; rung 0: DISPONIBILIDADE
LDNOT dp.dgm
ANDNOT dp.ndp
OUT dp.mdp
; rung 1: MODO DE FUNCIONAMENTO
LD dp.s_aut
OUT bmb.bits.s_aut
; rung 2: FUNCIONAMENTO AUTOMATICO
LD dp.s_aut
AND dp.mdp
OUT bmb.bits.cfa
; rung 3: RESET
LD dp.rst
SET bmb.bits.rst
RSET dp.rst
; rung 4: SINALIZADOR VERMELHO
LD bmb.bits.dgm
ORNOT dp.mdp
OUT dp.oms_red

## Function block fb_dp_bmb_agi
; FUNÇÃO DEPOSITO DE PRODUTO COM BOMBA/AGITADOR - Executa o funcionamento de um deposito de produto constituido por uma bomba e um agitador.
VAR_IN_OUT
  dp : s_deposito_p;  (* Dados do deposito *)
  bmb : s_equip;  (* Dados da bomba *)
  agi : s_equip;  (* Dados do agitador *)
END_VAR
VAR
  tm01 : TIMER;
  tm02 : TIMER;
  cfx_agi : BOOL;
END_VAR

